// TwinCAT 3 PLC project lcls_plc_113
// ProgramVersion: 3.1.4022.7
// libraries:
//   LCLS General, * (SLAC)
//   lcls-twincat-common-components-nrw, * (SLAC)
//   lcls-twincat-motion, * (SLAC)
//   lcls-twincat-optics, * (SLAC)
//   Tc2_Standard, * (Beckhoff Automation GmbH)
//   Tc2_System, * (Beckhoff Automation GmbH)
//   Tc3_Module, * (Beckhoff Automation GmbH)
// project tree:
//   / PlcTask.TcTTO
//   POUs/ FB_FlutterDetection.TcPOU, FB_TestTrigger.TcPOU, MAIN.TcPOU
// real-time tasks:
//   TASK PlcTask: cycle T#10ms, priority 20, ADS port 350
// motion (NC):
//   TASK NC-Task 1 SAF: cycle T#2ms, priority 4, ADS port 501
//   TASK NC-Task 1 SVB: cycle T#10ms, priority 8, ADS port 511
//   AXIS Axis 1 (id 1)
//     OtherSettings: AllowMotionCmdToSlave=true
//     encoder EncType=4
//       EncPara: MaxCount=#x0000ffff
//         SoftEndMinControl: Enable=true, Range=79
//         SoftEndMaxControl: Range=235
//         Inc: RefSoftSyncMask=#x0000ffff
//     drive DrvType=24
//       Analog: ScaleFactorActTorque=0.1
//       TimeComp: TaskDelayCycles=1
//     controller CtrType=1
//       CtrPara: PriorControlFactor=1
//         Observer: BandWidth=20
// I/O:
//   DEVICE Device 1 (EtherCAT), AmsNetId 172.21.148.88.2.1
//     Term 1 (EK1200) [EK1200-5000 EtherCAT Power supply (2A E-Bus)]
//       Term 2 (EL3052) [EL3052 2Ch. Ana. Input 4-20mA]
//       Term 3 (EL3202-0010) [EL3202-0010 2Ch. Ana. Input PT100 (RTD), High Precision]
//       Term 8 (EL7031)
//       Term 4 (EL9011) [EL9011 End Terminal]
// variable links:
//   (this object) <-> Device 1 (EtherCAT)/Term 1 (EK1200)/Term 8 (EL7031)
//     Drive/Inputs/In/nState1 @bit 3 <-> STM Status/Status/Error
//     Drive/Inputs/In/nState1 @bit 5 <-> STM Status/Status/Moving negative
//     Drive/Inputs/In/nState1 @bit 4 <-> STM Status/Status/Moving positive
//     Drive/Inputs/In/nState1 @bit 1 <-> STM Status/Status/Ready
//     Drive/Inputs/In/nState1 <-> STM Status/Status/Ready to enable
//     Drive/Inputs/In/nState1 @bit 6 <-> STM Status/Status/Torque reduced
//     Drive/Inputs/In/nState1 @bit 2 <-> STM Status/Status/Warning
//     Drive/Inputs/In/nState2 @bit 3 <-> STM Status/Status/Digital input 1
//     Drive/Inputs/In/nState2 @bit 4 <-> STM Status/Status/Digital input 2
//     Drive/Inputs/In/nState2 @bit 5 <-> STM Status/Status/Sync error
//     Drive/Inputs/In/nState2 @bit 7 <-> STM Status/Status/TxPDO Toggle
//     Drive/Inputs/In/nState4 @bit 1 <-> WcState/InputToggle
//     Drive/Inputs/In/nState4 <-> WcState/WcState
//     Drive/Outputs/Out/nCtrl1 <-> STM Control/Control/Enable
//     Drive/Outputs/Out/nCtrl1 @bit 2 <-> STM Control/Control/Reduce torque
//     Drive/Outputs/Out/nCtrl1 @bit 1 <-> STM Control/Control/Reset
//     Drive/Outputs/Out/nDataOut2[0] <-> STM Velocity/Velocity
//     Enc/Inputs/In/nDataIn1[0] <-> ENC Status compact/Counter value
//     Enc/Inputs/In/nDataIn2[0] <-> ENC Status compact/Latch value
//     Enc/Inputs/In/nState1 @bit 4 <-> ENC Status compact/Status/Counter overflow
//     Enc/Inputs/In/nState1 @bit 3 <-> ENC Status compact/Status/Counter underflow
//     Enc/Inputs/In/nState1 @bit 1 <-> ENC Status compact/Status/Latch extern valid
//     Enc/Inputs/In/nState1 @bit 2 <-> ENC Status compact/Status/Set counter done
//     Enc/Inputs/In/nState2 @bit 4 <-> ENC Status compact/Status/Status of extern latch
//     Enc/Inputs/In/nState2 @bit 5 <-> ENC Status compact/Status/Sync error
//     Enc/Inputs/In/nState2 @bit 7 <-> ENC Status compact/Status/TxPDO Toggle
//     Enc/Inputs/In/nState4 @bit 1 <-> WcState/InputToggle
//     Enc/Inputs/In/nState4 <-> WcState/WcState
//     Enc/Outputs/Out/nCtrl1 @bit 3 <-> ENC Control compact/Control/Enable latch extern on negative edge
//     Enc/Outputs/Out/nCtrl1 @bit 1 <-> ENC Control compact/Control/Enable latch extern on positive edge
//     Enc/Outputs/Out/nCtrl1 @bit 2 <-> ENC Control compact/Control/Set counter
//     Enc/Outputs/Out/nDataOut1[0] <-> ENC Control compact/Set counter value
//   lcls_plc_113 Instance <-> Device 1 (EtherCAT)/Term 1 (EK1200)/Term 3 (EL3202-0010)
//     PlcTask Inputs/MAIN.fbFlowMeter.iRaw <-> RTD Inputs Channel 1/Value
//     PlcTask Inputs/MAIN.fbTempSensor.iRaw <-> RTD Inputs Channel 1/Value
//   lcls_plc_113 Instance <-> NC-Task 1 SAF/Axes/Axis 1
//     PlcTask Inputs/MAIN.M1.Axis.NcToPlc <-> Outputs/ToPlc
//     PlcTask Outputs/MAIN.M1.Axis.PlcToNc <-> Inputs/FromPlc

CONFIGURATION lcls_plc_113
    RESOURCE PLC ON TwinCAT3
        TASK PlcTask(INTERVAL := T#10ms, PRIORITY := 20);
        PROGRAM MAIN WITH PlcTask : MAIN;
    END_RESOURCE
END_CONFIGURATION

// ---- POUs/MAIN.TcPOU
PROGRAM MAIN
VAR    
    {attribute 'pytmc' := '
        pv: RM113
    '}
    {attribute 'TcLinkTo' := '.iRaw := TIIB[Term 3 (EL3202-0010)]^RTD Inputs Channel 1^Value'}
    fbTempSensor : FB_TempSensor;
    fTemp : LREAL;
    
    {attribute 'pytmc' := '
        pv: RM113
    '}
    fbFlutterDet : FB_FlutterDetection;
    bTestFlip : BOOL;

    fbTrigTest : FB_TestTrigger;

    {attribute 'pytmc' := '
        pv: RM113:TST:MMS:Y
    '}
    M1 : ST_MotionStage := (fVelocity:=100.0, nEnableMode:=ENUM_StageEnableMode.ALWAYS, bPowerSelf:=True); // M1K2 Yleft
    fbMotionStage_m1 : FB_MotionStage;
    {attribute 'pytmc' := '
        pv: RM113:TST
    '}
    {attribute 'TcLinkTo' := '.iRaw := TIIB[Term 3 (EL3202-0010)]^RTD Inputs Channel 1^Value'}
    fbFlowMeter : FB_FDQ_FlowMeter;
END_VAR

fbTempSensor(fResolution:=0.01);

fTemp := fbTempSensor.fTemp;
fTemp := (9.0/5.0) * fTemp + 32;

fbFlutterDet(fPastTime:=T#5000ms, bVarToMonitor:=bTestFlip);
//fbTrigTest(bTestBool:=bTestFlip);

fbMotionStage_m1(stMotionStage:=M1);
fbFlowMeter();

END_PROGRAM

// ---- POUs/FB_FlutterDetection.TcPOU
FUNCTION_BLOCK FB_FlutterDetection
VAR_INPUT
    bVarToMonitor : BOOL;
    fPastTime : TIME := T#5000ms;
    nMaxFlipsAllowed : UINT := 10;
    bReset : BOOL;
END_VAR
VAR_OUTPUT
    {attribute 'pytmc' := '
        pv: TEST:OUT:1
        io: io
    '}
    bExceededFlipMax : BOOL;
END_VAR
VAR
    bInit : BOOL := FALSE;
    bLastVarValue : BOOL;
    nNumFlipped : UINT;
    tTimer : TON;
    rtReset : r_trig;
END_VAR

IF NOT bInit THEN
    bLastVarValue := bVarToMonitor;
    nNumFlipped := 0;
    bExceededFlipMax := FALSE;
    tTimer(IN:=FALSE);
    tTimer(IN:=TRUE, PT:=fPastTime); 
    bInit := TRUE;
END_IF    

rtReset(CLK:=bReset);

IF rtReset.Q THEN
    // re-initialize
    bInit := FALSE;
END_IF

bReset R= rtReset.Q;
tTimer();

IF tTimer.Q THEN
    IF nNumFlipped > nMaxFlipsAllowed THEN
        bExceededFlipMax := TRUE;
        // timer off, no need to count.
    ELSE
        nNumFlipped := 0;
        // reset timer
        tTimer(IN:=FALSE);
        tTimer(IN:=TRUE);
    END_IF    
END_IF

IF bLastVarValue <> bVarToMonitor THEN
    nNumFlipped := nNumFlipped +1;
    bLastVarValue := bVarToMonitor;
END_IF

END_FUNCTION_BLOCK

// ---- POUs/FB_TestTrigger.TcPOU
FUNCTION_BLOCK FB_TestTrigger
VAR_INPUT
    bTestBool : BOOL ;
END_VAR
VAR_OUTPUT
END_VAR
VAR
    rtRisingTrigger : r_trig;
END_VAR

rtRisingTrigger(CLK:=bTestBool);

END_FUNCTION_BLOCK
